{attribute 'linkalways'} 
{attribute 'no_explicit_call' := 'This FB is a CLASS and must be accessed using methods or properties'}
{attribute 'enable_dynamic_creation'}
FUNCTION_BLOCK FINAL LE_REAL EXTENDS Node
VAR
	in1 : _REAL(0.0);
	in2 : _REAL(0.0);
	out : _BOOL(FALSE);
END_VAR

METHOD PUBLIC Clone : I_Node
VAR
	pNode : POINTER TO LE_REAL;
END_VAR
pNode := __NEW(LE_REAL);
Clone := pNode^;
END_METHOD

METHOD FB_init : BOOL
VAR_INPUT
	bInitRetains : BOOL; // if TRUE, the retain variables are initialized (warm start / cold start)
	bInCopyCode : BOOL;  // if TRUE, the instance afterwards gets moved into the copy code (online change)
END_VAR
AddInput('in1',THIS^.in1);
AddInput('in2',THIS^.in2);
AddOutput('out', THIS^.out);
END_METHOD

METHOD PROTECTED OnExecute
VAR
END_VAR
out.Value := in1.Value <= in2.Value;
END_METHOD

END_FUNCTION_BLOCK

(* stored: Version 1.1.0.1, ProductVersion 3.1.4024.15
   POU LE_REAL: Id {6b57461b-05cd-43d9-baa1-b15a0f01fcc6}, SpecialFunc None
   Folder Constructor: Id {1dbe6258-0d92-4a2b-964d-336e369f4918}
   Method Clone: Id {5d8f4e2e-8fb8-41e1-ac23-a0e95da1a422}
   Method FB_init: Id {f7e20cc2-1325-489c-a3ab-a9471b5a66c0}
   Method OnExecute: Id {5f239603-230d-4f9a-b993-d8026a3af81b} *)
